ABB RobotStudio station: Test_1.rsstnx

Station Test_1 (saved by RobotStudio 22.2.9947.0)
Controller Controller2, task T_ROB1: task frame (RAPID world) sits at (0, 1513.97, 0) mm in the station
Controller Controller1, task T_ROB2: task frame (RAPID world) sits at (-438.37, 0, 0) mm in the station
Controller Controller1, task T_ROB1: task frame (RAPID world) sits at (-438.37, 0, 0) mm in the station
Controller Controller1
  mechanical unit ROB_1: IRB1410_5_144__01, 6 joints, base frame (0, 0, 0) mm
  mechanical unit ROB_2: IRB1600_6_120__02, 6 joints, base frame (2217.29, 0, 0) mm, rotated rx 0 ry 0 rz 180 deg
Controller Controller2
  mechanical unit ROB_1: IRB1410_5_144__01_4, 6 joints, base frame (0, 0, 0) mm
Layout (positions relative to the parent item):
  - IRB1410_5_144__01 [mechanism, from Robots\IRB1410_5_144_G_01.rslib] at (-438.37, 0, 0) mm; joint values [0.1041, -0.05, 0.3352, 0.0136, 0.0787, -0.0029] (rad or m)
  - 5 [part] at (473.91, 95.37, 916.54) mm, rotated rx 113.71 ry -0.59 rz 95.77 deg, size 500 x 81.5 x 287.9 mm
  - IRB1600_6_120__02 [mechanism, from Robots\IRB1600_6_120_G_02.rslib] at (1778.93, 0, 0) mm, rotated rx 0 ry 0 rz 180 deg; joint values [0.0137, 0.1111, -0.2443, 0.4107, 0.7052, -0.6246] (rad or m)
  - MyTool [mechanism, from Training Objects\myTool.rslib] at (927.69, -28.46, 1006.53) mm, rotated rx -164.64 ry 59.61 rz 35.69 deg
  - IRB1410_5_144__01_4 [mechanism, from Robots\IRB1410_5_144_G_01.rslib] at (0, 1513.97, 0) mm; joint values [0.0638, -0.1484, 0.4395, -0.0887, 0.4634, 0.1294] (rad or m)
  - Platform_3 [part] at (760.02, 1413.37, 0) mm, size 500 x 500 x 500 mm
  - workpiece_2 [part] at (760.02, 1413.37, 518.46) mm, size 400 x 300 x 80 mm
  - MyTool_3 [mechanism, from Training Objects\myTool.rslib] at (815.19, 1562.66, 804.07) mm, rotated rx -180 ry 38.41 rz -180 deg
  - Fence_2500 [graphiccomponentgroup, from Equipment\Fence_2500.rslib] at (2847.99, 1784.44, 0) mm, rotated rx 0 ry 0 rz -179.62 deg
    - Body 1 [part, from Equipment\Fence_2500.rslib]
    - Body 2 [part, from Equipment\Fence_2500.rslib]
  - Fence_2501 [graphiccomponentgroup, from Equipment\Fence_2500.rslib] at (-975.12, 1757.99, 0) mm
    - Body 1 [part, from Equipment\Fence_2500.rslib]
    - Body 2 [part, from Equipment\Fence_2500.rslib]
  - Fence_2502 [graphiccomponentgroup, from Equipment\Fence_2500.rslib] at (-1382.49, -1040.39, 0) mm
    - Body 1 [part, from Equipment\Fence_2500.rslib]
    - Body 2 [part, from Equipment\Fence_2500.rslib]
  - Fence_2503 [graphiccomponentgroup, from Equipment\Fence_2500.rslib] at (-1014.21, -942.62, 0) mm, rotated rx 0 ry 0 rz -88.71 deg
    - Body 1 [part, from Equipment\Fence_2500.rslib]
    - Body 2 [part, from Equipment\Fence_2500.rslib]
  - Fence_740 [graphiccomponentgroup, from Equipment\Fence_740.rslib] at (2248.98, -1272.37, 0) mm, rotated rx 0 ry 0 rz 89.25 deg
    - Body 1 [part, from Equipment\Fence_740.rslib]
    - Body 2 [part, from Equipment\Fence_740.rslib]
Attachment: 5 is attached to IRB1410_5_144__01 / Link6
Attachment: MyTool is attached to IRB1600_6_120__02 / Link6
Attachment: workpiece_2 is attached to Platform_3
Attachment: MyTool_3 is attached to IRB1410_5_144__01_4 / Link6
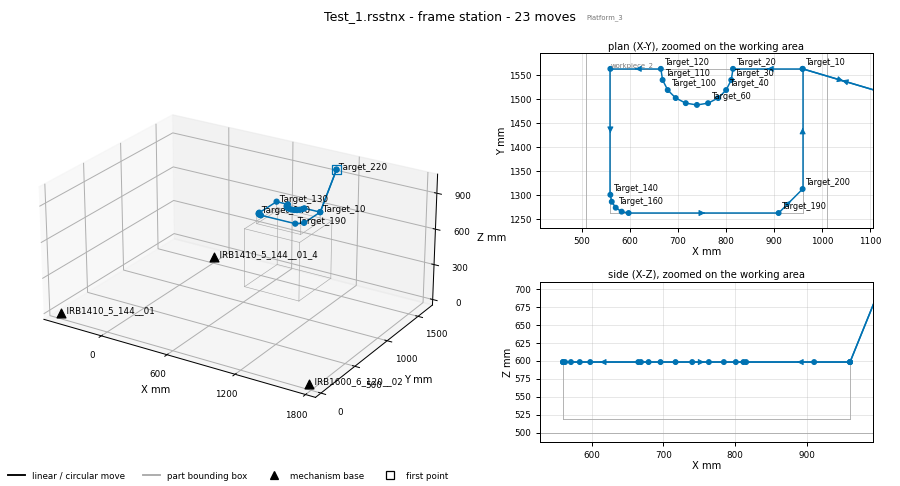
[picture p0: tool path of Test_1.rsstnx in frame station, 23 of 40 moves have a stored position in this frame; points joined in program order, loops and branches not executed]
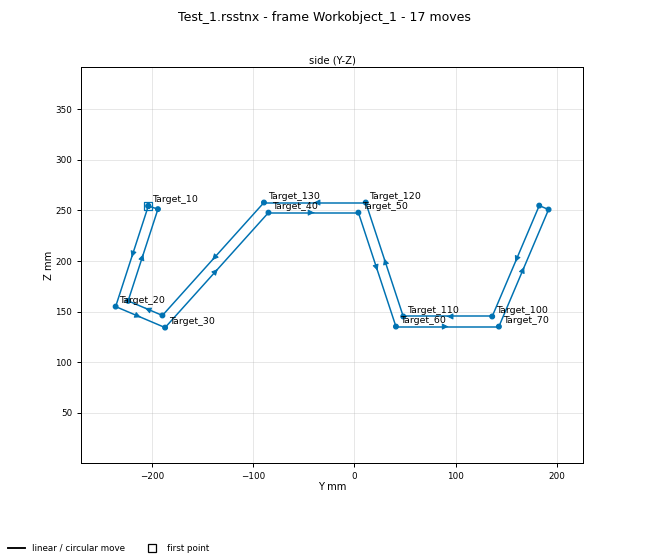
[picture p1: tool path of Test_1.rsstnx in frame Workobject_1, 17 of 40 moves have a stored position in this frame; points joined in program order, loops and branches not executed]
Targets, tools, work objects and paths stored in the station, written as RAPID:
! task T_ROB2
MODULE CalibData
  PERS tooldata MyTool:=[TRUE,[[31.792631019,0,229.638935148],[0.945518576,0,0.325568154,0]],[1,[0,0,1],[1,0,0,0],0,0,0]];
  TASK PERS wobjdata Workobject_1:=[FALSE,FALSE,"ROB_1",[[1208.667982233,-259.786332667,794.484345512],[0.696589706,0.153679796,0.148972451,0.684801074]],[[0,0,0],[1,0,0,0]]];
ENDMODULE

! task T_ROB2
MODULE Module1
  CONST robtarget Target_10:=[[-60,-203.867068409,254.436574641],[0.11061582,0.698407699,0.110615923,0.698394548],[0,0,0,0],[9E+09,9E+09,9E+09,9E+09,9E+09,9E+09]];
  CONST robtarget Target_20:=[[-59.999999999,-236.184577372,154.97350934],[0.11061582,0.698407699,0.110615923,0.698394548],[0,0,0,0],[9E+09,9E+09,9E+09,9E+09,9E+09,9E+09]];
  CONST robtarget Target_30:=[[-60,-187.258965467,134.205819219],[0.11061582,0.698407699,0.110615923,0.698394548],[0,0,0,0],[9E+09,9E+09,9E+09,9E+09,9E+09,9E+09]];
  CONST robtarget Target_40:=[[-60,-85.044509222,247.891489668],[0.11061582,0.698407699,0.110615923,0.698394548],[0,0,0,0],[9E+09,9E+09,9E+09,9E+09,9E+09,9E+09]];
  CONST robtarget Target_50:=[[-59.999999999,3.878988935,247.891489668],[0.11061582,0.698407699,0.110615923,0.698394548],[0,0,0,0],[9E+09,9E+09,9E+09,9E+09,9E+09,9E+09]];
  CONST robtarget Target_60:=[[-60,41.014913739,135.202937257],[0.11061582,0.698407699,0.110615923,0.698394548],[0,0,0,0],[9E+09,9E+09,9E+09,9E+09,9E+09,9E+09]];
  CONST robtarget Target_70:=[[-60,142.810926639,135.202937257],[0.11061582,0.698407699,0.110615923,0.698394548],[0,0,0,0],[9E+09,9E+09,9E+09,9E+09,9E+09,9E+09]];
  CONST robtarget Target_80:=[[-60,191.937475674,250.937834026],[0.11061582,0.698407699,0.110615923,0.698394548],[0,0,0,0],[9E+09,9E+09,9E+09,9E+09,9E+09,9E+09]];
  CONST robtarget Target_90:=[[-60.000000001,182.732427139,254.845145311],[0.11061582,0.698407699,0.110615923,0.698394548],[0,0,0,0],[9E+09,9E+09,9E+09,9E+09,9E+09,9E+09]];
  CONST robtarget Target_100:=[[-60,136.192071026,145.202937257],[0.11061582,0.698407699,0.110615923,0.698394548],[0,0,0,0],[9E+09,9E+09,9E+09,9E+09,9E+09,9E+09]];
  CONST robtarget Target_110:=[[-60,48.248472324,145.202937257],[0.11061582,0.698407699,0.110615923,0.698394548],[0,0,0,0],[9E+09,9E+09,9E+09,9E+09,9E+09,9E+09]];
  CONST robtarget Target_120:=[[-60,11.112547519,257.891489669],[0.11061582,0.698407699,0.110615923,0.698394548],[0,0,0,0],[9E+09,9E+09,9E+09,9E+09,9E+09,9E+09]];
  CONST robtarget Target_130:=[[-60.000000001,-89.501123873,257.891489669],[0.11061582,0.698407699,0.110615923,0.698394548],[0,0,0,0],[9E+09,9E+09,9E+09,9E+09,9E+09,9E+09]];
  CONST robtarget Target_140:=[[-60,-189.92256825,146.200055295],[0.11061582,0.698407699,0.110615923,0.698394548],[0,0,0,0],[9E+09,9E+09,9E+09,9E+09,9E+09,9E+09]];
  CONST robtarget Target_150:=[[-60,-223.842393157,160.598166739],[0.11061582,0.698407699,0.110615923,0.698394548],[0,0,0,0],[9E+09,9E+09,9E+09,9E+09,9E+09,9E+09]];
  CONST robtarget Target_160:=[[-60,-194.356503245,251.346404697],[0.11061582,0.698407699,0.110615923,0.698394548],[0,0,0,0],[9E+09,9E+09,9E+09,9E+09,9E+09,9E+09]];
  CONST robtarget Target_170:=[[-60,-203.867068409,254.436574641],[0.11061582,0.698407699,0.110615923,0.698394548],[0,0,0,0],[9E+09,9E+09,9E+09,9E+09,9E+09,9E+09]];
  CONST robtarget Target_180:=[[1184.687388799,-1891.987131155,604.132758068],[0,0,1,0],[0,0,0,0],[9E+09,9E+09,9E+09,9E+09,9E+09,9E+09]];
  CONST robtarget Target_190:=[[1496.687388799,-1891.987131155,604.132758068],[0,0,1,0],[0,0,0,0],[9E+09,9E+09,9E+09,9E+09,9E+09,9E+09]];
  CONST robtarget Target_200:=[[1546.687388799,-1841.987131155,604.132758068],[0,0,1,0],[0,0,0,0],[9E+09,9E+09,9E+09,9E+09,9E+09,9E+09]];
  CONST robtarget Target_210:=[[1546.687388799,-1591.987131155,604.132758068],[0,0,1,0],[0,0,0,0],[9E+09,9E+09,9E+09,9E+09,9E+09,9E+09]];
  CONST robtarget Target_220:=[[1401.855957026,-1591.987131155,604.132758068],[0,0,1,0],[0,0,0,0],[9E+09,9E+09,9E+09,9E+09,9E+09,9E+09]];
  CONST robtarget Target_230:=[[1398.18107059,-1615.189450957,604.132758068],[0,0,1,0],[0,0,0,0],[9E+09,9E+09,9E+09,9E+09,9E+09,9E+09]];
  CONST robtarget Target_240:=[[1387.516134771,-1636.120566036,604.132758068],[0,0,1,0],[0,0,0,0],[9E+09,9E+09,9E+09,9E+09,9E+09,9E+09]];
  CONST robtarget Target_250:=[[1370.905107793,-1652.731593014,604.132758068],[0,0,1,0],[0,0,0,0],[9E+09,9E+09,9E+09,9E+09,9E+09,9E+09]];
  CONST robtarget Target_260:=[[1349.973992714,-1663.396528833,604.132758068],[0,0,1,0],[0,0,0,0],[9E+09,9E+09,9E+09,9E+09,9E+09,9E+09]];
  CONST robtarget Target_270:=[[1326.771672912,-1667.071415269,604.132758068],[0,0,1,0],[0,0,0,0],[9E+09,9E+09,9E+09,9E+09,9E+09,9E+09]];
  CONST robtarget Target_280:=[[1303.569353111,-1663.396528833,604.132758068],[0,0,1,0],[0,0,0,0],[9E+09,9E+09,9E+09,9E+09,9E+09,9E+09]];
  CONST robtarget Target_290:=[[1282.638238032,-1652.731593014,604.132758068],[0,0,1,0],[0,0,0,0],[9E+09,9E+09,9E+09,9E+09,9E+09,9E+09]];
  CONST robtarget Target_300:=[[1266.027211054,-1636.120566036,604.132758068],[0,0,1,0],[0,0,0,0],[9E+09,9E+09,9E+09,9E+09,9E+09,9E+09]];
  CONST robtarget Target_310:=[[1255.362275235,-1615.189450957,604.132758068],[0,0,1,0],[0,0,0,0],[9E+09,9E+09,9E+09,9E+09,9E+09,9E+09]];
  CONST robtarget Target_320:=[[1251.687388799,-1591.987131155,604.132758068],[0,0,1,0],[0,0,0,0],[9E+09,9E+09,9E+09,9E+09,9E+09,9E+09]];
  CONST robtarget Target_330:=[[1146.687388799,-1591.987131155,604.132758068],[0,0,1,0],[0,0,0,0],[9E+09,9E+09,9E+09,9E+09,9E+09,9E+09]];
  CONST robtarget Target_340:=[[1146.687388799,-1853.987131155,604.132758068],[0,0,1,0],[0,0,0,0],[9E+09,9E+09,9E+09,9E+09,9E+09,9E+09]];
  CONST robtarget Target_350:=[[1149.579966564,-1868.529101585,604.132758068],[0,0,1,0],[0,0,0,0],[9E+09,9E+09,9E+09,9E+09,9E+09,9E+09]];
  CONST robtarget Target_360:=[[1157.817331114,-1880.85718884,604.132758068],[0,0,1,0],[0,0,0,0],[9E+09,9E+09,9E+09,9E+09,9E+09,9E+09]];
  CONST robtarget Target_370:=[[1170.145418369,-1889.094553391,604.132758068],[0,0,1,0],[0,0,0,0],[9E+09,9E+09,9E+09,9E+09,9E+09,9E+09]];
  CONST robtarget Target_380:=[[1184.687388799,-1891.987131155,604.132758068],[0,0,1,0],[0,0,0,0],[9E+09,9E+09,9E+09,9E+09,9E+09,9E+09]];
  PROC Path_10()
    MoveL Target_10,v1000,z100,MyTool\WObj:=Workobject_1;
    MoveL Target_20,v1000,z100,MyTool\WObj:=Workobject_1;
    MoveL Target_30,v1000,z100,MyTool\WObj:=Workobject_1;
    MoveL Target_40,v1000,z100,MyTool\WObj:=Workobject_1;
    MoveL Target_50,v1000,z100,MyTool\WObj:=Workobject_1;
    MoveL Target_60,v1000,z100,MyTool\WObj:=Workobject_1;
    MoveL Target_70,v1000,z100,MyTool\WObj:=Workobject_1;
    MoveL Target_80,v1000,z100,MyTool\WObj:=Workobject_1;
    MoveL Target_90,v1000,z100,MyTool\WObj:=Workobject_1;
    MoveL Target_100,v1000,z100,MyTool\WObj:=Workobject_1;
    MoveL Target_110,v1000,z100,MyTool\WObj:=Workobject_1;
    MoveL Target_120,v1000,z100,MyTool\WObj:=Workobject_1;
    MoveL Target_130,v1000,z100,MyTool\WObj:=Workobject_1;
    MoveL Target_140,v1000,z100,MyTool\WObj:=Workobject_1;
    MoveL Target_150,v1000,z100,MyTool\WObj:=Workobject_1;
    MoveL Target_160,v1000,z100,MyTool\WObj:=Workobject_1;
    MoveL Target_170,v1000,z100,MyTool\WObj:=Workobject_1;
  ENDPROC
ENDMODULE

! task T_ROB1
MODULE CalibData
  PERS tooldata MyTool:=[TRUE,[[31.792631019,0,229.638935148],[0.945518576,0,0.325568154,0]],[1,[0,0,1],[1,0,0,0],0,0,0]];
  TASK PERS wobjdata Workobject_3:=[FALSE,TRUE,"",[[1010.021,149.404,500],[0,0,0,1]],[[0,0,0],[1,0,0,0]]];
ENDMODULE

! task T_ROB1
MODULE Module1
  CONST robtarget Target_10:=[[49.999618624,100.00021347,98.459574342],[0,1,0,0],[0,0,0,0],[9E+09,9E+09,9E+09,9E+09,9E+09,9E+09]];
  CONST robtarget Target_20:=[[194.831050397,100.00021347,98.459574342],[0,1,0,0],[0,0,0,0],[9E+09,9E+09,9E+09,9E+09,9E+09,9E+09]];
  CONST robtarget Target_30:=[[198.505936833,123.202533272,98.459574342],[0,1,0,0],[0,0,0,0],[9E+09,9E+09,9E+09,9E+09,9E+09,9E+09]];
  CONST robtarget Target_40:=[[209.170872653,144.133648351,98.459574342],[0,1,0,0],[0,0,0,0],[9E+09,9E+09,9E+09,9E+09,9E+09,9E+09]];
  CONST robtarget Target_50:=[[225.78189963,160.744675329,98.459574342],[0,1,0,0],[0,0,0,0],[9E+09,9E+09,9E+09,9E+09,9E+09,9E+09]];
  CONST robtarget Target_60:=[[246.713014709,171.409611148,98.459574342],[0,1,0,0],[0,0,0,0],[9E+09,9E+09,9E+09,9E+09,9E+09,9E+09]];
  CONST robtarget Target_70:=[[269.915334511,175.084497584,98.459574342],[0,1,0,0],[0,0,0,0],[9E+09,9E+09,9E+09,9E+09,9E+09,9E+09]];
  CONST robtarget Target_80:=[[293.117654312,171.409611148,98.459574342],[0,1,0,0],[0,0,0,0],[9E+09,9E+09,9E+09,9E+09,9E+09,9E+09]];
  CONST robtarget Target_90:=[[314.048769391,160.744675329,98.459574342],[0,1,0,0],[0,0,0,0],[9E+09,9E+09,9E+09,9E+09,9E+09,9E+09]];
  CONST robtarget Target_100:=[[330.659796369,144.133648351,98.459574342],[0,1,0,0],[0,0,0,0],[9E+09,9E+09,9E+09,9E+09,9E+09,9E+09]];
  CONST robtarget Target_110:=[[341.324732188,123.202533272,98.459574342],[0,1,0,0],[0,0,0,0],[9E+09,9E+09,9E+09,9E+09,9E+09,9E+09]];
  CONST robtarget Target_120:=[[344.999618624,100.00021347,98.459574342],[0,1,0,0],[0,0,0,0],[9E+09,9E+09,9E+09,9E+09,9E+09,9E+09]];
  CONST robtarget Target_130:=[[449.999618624,100.00021347,98.459574342],[0,1,0,0],[0,0,0,0],[9E+09,9E+09,9E+09,9E+09,9E+09,9E+09]];
  CONST robtarget Target_140:=[[449.999618624,362.00021347,98.459574342],[0,1,0,0],[0,0,0,0],[9E+09,9E+09,9E+09,9E+09,9E+09,9E+09]];
  CONST robtarget Target_150:=[[447.10704086,376.5421839,98.459574342],[0,1,0,0],[0,0,0,0],[9E+09,9E+09,9E+09,9E+09,9E+09,9E+09]];
  CONST robtarget Target_160:=[[438.869676309,388.870271155,98.459574342],[0,1,0,0],[0,0,0,0],[9E+09,9E+09,9E+09,9E+09,9E+09,9E+09]];
  CONST robtarget Target_170:=[[426.541589054,397.107635706,98.459574342],[0,1,0,0],[0,0,0,0],[9E+09,9E+09,9E+09,9E+09,9E+09,9E+09]];
  CONST robtarget Target_180:=[[411.999618624,400.00021347,98.459574342],[0,1,0,0],[0,0,0,0],[9E+09,9E+09,9E+09,9E+09,9E+09,9E+09]];
  CONST robtarget Target_190:=[[99.999618624,400.00021347,98.459574342],[0,1,0,0],[0,0,0,0],[9E+09,9E+09,9E+09,9E+09,9E+09,9E+09]];
  CONST robtarget Target_200:=[[49.999618624,350.00021347,98.459574342],[0,1,0,0],[0,0,0,0],[9E+09,9E+09,9E+09,9E+09,9E+09,9E+09]];
  CONST robtarget Target_210:=[[49.999618624,100.00021347,98.459574342],[0,1,0,0],[0,0,0,0],[9E+09,9E+09,9E+09,9E+09,9E+09,9E+09]];
  CONST robtarget Target_220:=[[-116.567995348,149.404,510.14730631],[0,0.981627183,0,-0.190808996],[0,-1,0,0],[9E+09,9E+09,9E+09,9E+09,9E+09,9E+09]];
  PROC Path_10()
    MoveL Target_220,v1000,z100,MyTool\WObj:=Workobject_3;
    MoveL Target_10,v1000,z100,MyTool\WObj:=Workobject_3;
    MoveL Target_20,v1000,z100,MyTool\WObj:=Workobject_3;
    MoveL Target_30,v1000,z100,MyTool\WObj:=Workobject_3;
    MoveL Target_40,v1000,z100,MyTool\WObj:=Workobject_3;
    MoveL Target_50,v1000,z100,MyTool\WObj:=Workobject_3;
    MoveL Target_60,v1000,z100,MyTool\WObj:=Workobject_3;
    MoveL Target_70,v1000,z100,MyTool\WObj:=Workobject_3;
    MoveL Target_80,v1000,z100,MyTool\WObj:=Workobject_3;
    MoveL Target_90,v1000,z100,MyTool\WObj:=Workobject_3;
    MoveL Target_100,v1000,z100,MyTool\WObj:=Workobject_3;
    MoveL Target_110,v1000,z100,MyTool\WObj:=Workobject_3;
    MoveL Target_120,v1000,z100,MyTool\WObj:=Workobject_3;
    MoveL Target_130,v1000,z100,MyTool\WObj:=Workobject_3;
    MoveL Target_140,v1000,z100,MyTool\WObj:=Workobject_3;
    MoveL Target_150,v1000,z100,MyTool\WObj:=Workobject_3;
    MoveL Target_160,v1000,z100,MyTool\WObj:=Workobject_3;
    MoveL Target_170,v1000,z100,MyTool\WObj:=Workobject_3;
    MoveL Target_180,v1000,z100,MyTool\WObj:=Workobject_3;
    MoveL Target_190,v1000,z100,MyTool\WObj:=Workobject_3;
    MoveL Target_200,v1000,z100,MyTool\WObj:=Workobject_3;
    MoveL Target_210,v1000,z100,MyTool\WObj:=Workobject_3;
    MoveL Target_220,v1000,z100,MyTool\WObj:=Workobject_3;
  ENDPROC
ENDMODULE

